{attribute 'qualified_only'}
{attribute 'strict'}
TYPE EFeedbackMsgAttenuationFW212C :
(
	CheckConnectionMsg := 10,
    PositionMsg,
    PositionCountMsg,
    IdMsg,
    CustomMsg
);
END_TYPE

(* stored: Version 1.1.0.1, ProductVersion 3.1.4024.4
   DUT EFeedbackMsgAttenuationFW212C: Id {f1e93c99-4c55-41eb-a2b5-4489e2258cf5} *)
